// SIMATIC STEP 7 (V5.x) project blinkerPLC
// CPU: CPU 315-2 DP
// CPU: CPU 315-2 DP
// station: Hardware
// station: SIMATIC 300(1)
// station: P_ADR_BUS
// station: P_ADR_BUS
// station: Hardware
// station: SIMATIC 300(2)
// program: S7 Program(1)
// program: S7 Program(2)

SYMBOL_TABLE
"COUNTER"	C 0	COUNTER
"START_BUTTON"	I 0.0	BOOL
"STOP_BUTTON"	I 0.1	BOOL
"SETBUTTON"	I 0.2	BOOL
"MASTERBIT"	M 0.0	BOOL
"STOPBIT"	M 0.1	BOOL
"COUNTERACC"	MW 1	WORD
"MOTOR1"	Q 4.0	BOOL
"MOTOR2"	Q 4.1	BOOL
"TIMER_MOTOR_1"	T 0	TIMER
"TIMER_MOTOR2"	T 1	TIMER
END_SYMBOL_TABLE

ORGANIZATION_BLOCK OB 1
TITLE = "Main Program Sweep (Cycle)"
VERSION : 0.1
VAR_TEMP
  OB1_EV_CLASS : BYTE ;	//Bits 0-3 = 1 (Coming event), Bits 4-7 = 1 (Event class 1)
  OB1_SCAN_1 : BYTE ;	//1 (Cold restart scan 1 of OB 1), 3 (Scan 2-n of OB 1)
  OB1_PRIORITY : BYTE ;	//Priority of OB Execution
  OB1_OB_NUMBR : BYTE ;	//1 (Organization block 1, OB1)
  OB1_RESERVED_1 : BYTE ;	//Reserved for system
  OB1_RESERVED_2 : BYTE ;	//Reserved for system
  OB1_PREV_CYCLE : INT ;	//Cycle time of previous OB1 scan (milliseconds)
  OB1_MIN_CYCLE : INT ;	//Minimum cycle time of OB1 (milliseconds)
  OB1_MAX_CYCLE : INT ;	//Maximum cycle time of OB1 (milliseconds)
  OB1_DATE_TIME : DATE_AND_TIME ;	//Date and time OB1 started
END_VAR
BEGIN
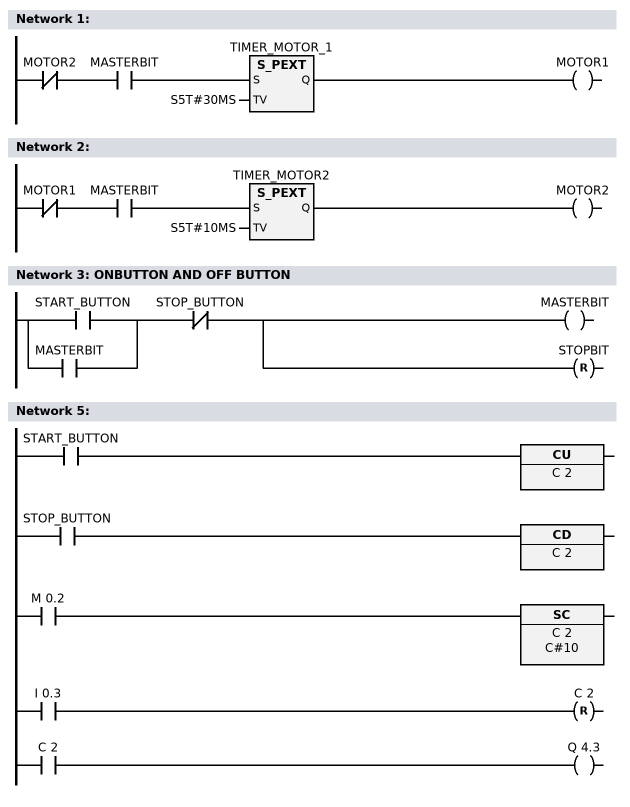
NETWORK
TITLE =
      AN    "MOTOR2";
      A     "MASTERBIT";
      L     S5T#30MS;
      SE    "TIMER_MOTOR_1";
      NOP   0;
      NOP   0;
      NOP   0;
      A     "TIMER_MOTOR_1";
      =     "MOTOR1";
NETWORK
TITLE =
      AN    "MOTOR1";
      A     "MASTERBIT";
      L     S5T#10MS;
      SE    "TIMER_MOTOR2";
      NOP   0;
      NOP   0;
      NOP   0;
      A     "TIMER_MOTOR2";
      =     "MOTOR2";
NETWORK
TITLE = ONBUTTON AND OFF BUTTON
      A(;
      O     "START_BUTTON";
      O     "MASTERBIT";
      );
      AN    "STOP_BUTTON";
      =     "MASTERBIT";
      R     "STOPBIT";
NETWORK
TITLE = COUNTERS
//THe up counter just set the PV and watch it start from 0 to the PV
//the down counter set the PV then SET the counter and let it count down to zero
      O     "MOTOR2";
      O     "MOTOR1";
      =     L 20.0;
      A(;
      A     L 20.0;
      CU    "COUNTER";
      BLD   101;
      A     "SETBUTTON";
      L     C#0;
      S     "COUNTER";
      A     "STOP_BUTTON";
      R     "COUNTER";
      L     "COUNTER";
      T     "COUNTERACC";
      NOP   0;
      A     "COUNTER";
      );
      A(;
      L     "COUNTERACC";
      L     100;
      >I;
      );
      R     "MASTERBIT";
      S     "STOPBIT";
      A     L 20.0;
      CD    C 1;
      BLD   101;
      A     "MASTERBIT";
      L     C#100;
      S     C 1;
      A     "STOP_BUTTON";
      R     C 1;
      NOP   0;
      NOP   0;
      NOP   0;
NETWORK
TITLE =
      A     "START_BUTTON";
      CU    C 2;
      A     "STOP_BUTTON";
      CD    C 2;
      A     M 0.2;
      L     C#10;
      S     C 2;
      A     I 0.3;
      R     C 2;
      NOP   0;
      NOP   0;
      A     C 2;
      =     Q 4.3;
END_ORGANIZATION_BLOCK

ORGANIZATION_BLOCK OB 1
VERSION : 0.1
BEGIN
// (block stored without names or comments; labels and parameter names are numbered)
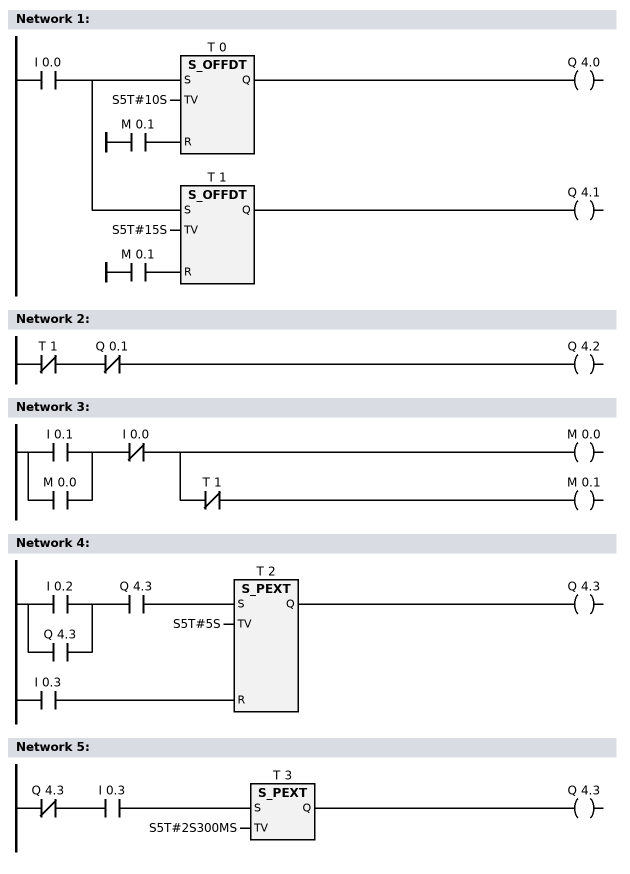
NETWORK
TITLE =
      A     I 0.0;
      =     L 20.0;
      A     L 20.0;
      L     S5T#10S;
      SF    T 0;
      A     M 0.1;
      R     T 0;
      NOP   0;
      NOP   0;
      A     T 0;
      =     Q 4.0;
      A     L 20.0;
      L     S5T#15S;
      SF    T 1;
      A     M 0.1;
      R     T 1;
      NOP   0;
      NOP   0;
      A     T 1;
      =     Q 4.1;
NETWORK
TITLE =
      AN    T 1;
      AN    Q 0.1;
      =     Q 4.2;
NETWORK
TITLE =
      A(;
      O     I 0.1;
      O     M 0.0;
      );
      AN    I 0.0;
      =     L 20.0;
      A     L 20.0;
      BLD   102;
      =     M 0.0;
      A     L 20.0;
      AN    T 1;
      =     M 0.1;
NETWORK
TITLE =
      A(;
      O     I 0.2;
      O     Q 4.3;
      );
      A     Q 4.3;
      L     S5T#5S;
      SE    T 2;
      A     I 0.3;
      R     T 2;
      NOP   0;
      NOP   0;
      A     T 2;
      =     Q 4.3;
NETWORK
TITLE =
      AN    Q 4.3;
      A     I 0.3;
      L     S5T#2S300MS;
      SE    T 3;
      NOP   0;
      NOP   0;
      NOP   0;
      A     T 3;
      =     Q 4.3;
END_ORGANIZATION_BLOCK
